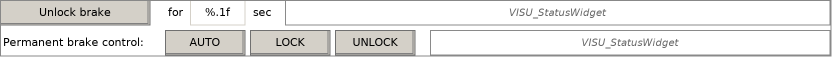
VISUALIZATION VISU_Axes_Commands_Brake  // 832x57
VAR_IN_OUT
    unlockBrake : AxesUnlockBrakeProcess;
    setBrake : SetBrakeProcess;
    unlockBrakeStatus : StatusWidget;
    setBrakeStatus : StatusWidget;
END_VAR
    Button (0,0 150x25), "Unlock brake", input disabled if: unlockBrake.statuses.enabledStatus.disabled
        OnMouseClick: execute { unlockBrake.do_request := TRUE; }
    Frame (285,0 545x25)
        shows VISU_StatusWidget(widget := unlockBrakeStatus)
    Textfield (190,0 55x25), "%.1f", text variable: unlockBrake.set.seconds
        OnMouseClick: write the text variable via VisuDialogs.Numpad
    Label (165,0 30x25), "for"
    Label (245,0 35x25), "sec"
    Button (165,30 80x25), "AUTO", input disabled if: setBrake.statuses.enabledStatus.disabled
        OnMouseClick: execute { setBrake.request(DriveBrakeStates.BRAKE_AUTOMATIC); }
    Button (250,30 80x25), "LOCK", input disabled if: setBrake.statuses.enabledStatus.disabled
        OnMouseClick: execute { setBrake.request(DriveBrakeStates.BRAKE_FORCE_LOCK); }
    Button (335,30 80x25), "UNLOCK", input disabled if: setBrake.statuses.enabledStatus.disabled
        OnMouseClick: execute { setBrake.request(DriveBrakeStates.BRAKE_FORCE_UNLOCK); }
    Frame (430,30 400x25)
        shows VISU_StatusWidget(widget := setBrakeStatus)
    Label (0,30 165x25), "Permanent brake control:"
END_VISUALIZATION

(* stored: Version 1.1.0.1, ProductVersion 3.1.4019.2
   Visu VISU_Axes_Commands_Brake: Id {11e1d53e-adf4-4f1d-9f08-7ce0659c0657} *)
